PROGRAM Initialiseren
VAR
	timer1: ton;
END_VAR

IF GVL.Initialisatie_voltooid = FALSE AND GVL.Initialiseren =TRUE THEN
	Simulatie_Invoer();
END_IF

			
			IF GVL.ZaagLengte = GVL.HuidigePositieAanvoer THEN 
			GVL.Initialisatie_voltooid := TRUE;	
			GVL.Initialiseren:=FALSE;	
			END_IF

END_PROGRAM

(* stored: Version 1.1.0.1, ProductVersion 3.1.4024.12
   POU Initialiseren: Id {50253b7d-fc8b-4a12-9fbd-309ed75f9929}, SpecialFunc None *)
